# B&R Automation Studio project CoffeeMachine
Automation Studio 4.12.3.127 SP; Default project; technology packages: Acp10Arnc0 5.16.2, mappSafety 5.16.0, mappView 5.16.1

## Configuration ARX

CPU 4PPC30.043F-22B, AutomationRuntime B4.93, Build 4.1.2, Vc V4.72.6

### Hardware
```
4PPC30_043F_22B : 4PPC30.043F-22B v1.1.3.0
  Connector IF3:
    ActivateDevice = 1
  ConfigurationID = CoffeeMachine_ARX
  TimerDeviceType = SWIOTIMER
  Cyclic1Duration = 10000
  Cyclic1Tolerance = 10000
  Cyclic2Duration = 20000
  Cyclic2Tolerance = 20000
  Cyclic3Duration = 50000
  Cyclic3Tolerance = 50000
  Cyclic4Duration = 100000
  Cyclic4Tolerance = 100000
  Cyclic5Duration = 200000
  Cyclic5Tolerance = 200000
  Cyclic6Duration = 500000
  Cyclic6Tolerance = 500000
  Cyclic7Duration = 1000000
  Cyclic7Tolerance = 1000000
  Cyclic8Duration = 10000
  Cyclic8Tolerance = 30000000
  FileDevice1
  FileDeviceName1 = USER
  FileDevicePath1 = USER_PATH
  KeyMappingFile = VC\4PPC30_043F_22B.dis
```

## Configuration Simulation

CPU , AutomationRuntime B4.93, Build 4.1.2, Safety 0.0, Vc V4.72.6

### Hardware
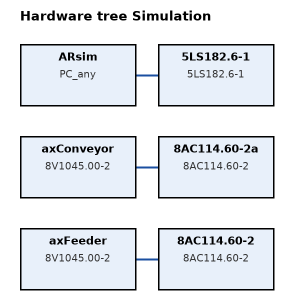
```
5LS182.6-1 : 5LS182.6-1 v1.3.1.0  [SL -> ARsim.SL1]
  Connector IF1:
    DNAConfiguration = manual
8AC114.60-2 : 8AC114.60-2 v1.0.0.8  [SS -> axFeeder.SS1; PLK1 -> 5LS182.6-1.IF1 (NodeNumber=1) [Cable Type=PowerlinkCable, Length=10, Version=1.0.0.3]; PLK2 -> 8AC114.60-2a.PLK1 (NodeNumber=1) [Cable Type=PowerlinkCable, Length=10, Version=1.0.0.3]]
8AC114.60-2a : 8AC114.60-2 v1.0.0.8  [SS -> axConveyor.SS1; PLK1 -> 8AC114.60-2.PLK2 (NodeNumber=2) [Cable Type=PowerlinkCable, Length=10, Version=1.0.0.3]]
ARsim : PC_any v1.1.1.0 (OrderNumber=PC)
  Connector IF3:
    Vnc1
    VncVcObjectName1 = Visu
    VncAuthentication1 = 1
    VncPasswordViewOnly1 = v
    VncPasswordViewControl1 = c
    VncRefreshRate1 = 200
    VncTitle1 = VNC - B&R Coffee Machine
  PreserveNonVolatileSystemSettings = 0
  BRObjects = 450
  XLinkUseDefault = 0
  Cyclic1Duration = 10000
  Cyclic1Tolerance = 0
  Cyclic2Duration = 200000
  Cyclic2Tolerance = 10000000
  Cyclic3Duration = 500000
  Cyclic3Tolerance = 10000000
  Cyclic4Duration = 1000000
  Cyclic4Tolerance = 10000000
  Cyclic5Duration = 2000000
  Cyclic5Tolerance = 10000000
  Cyclic6Duration = 3000000
  Cyclic6Tolerance = 12000000
  Cyclic7Duration = 4000000
  Cyclic7Tolerance = 12000000
  Cyclic8Duration = 5000000
  Cyclic8Tolerance = 30000000
  EthernetHostName = AR000CoffeeMachine
  ActivateOpcUa = 1
axConveyor : 8V1045.00-2 v2.2.0.0
  Simulate = standard
axFeeder : 8V1045.00-2 v2.2.0.0
  Simulate = standard
```

## Configuration T50_X20CP1586mcSim

### Task classes (Cpu.sw)
```
Cyclic#1 (cycle 2000 us, tolerance 0 us):
  mainlogic <- mainlogic.prg
  feeder <- FeederArm.feeder.prg
  conveyor <- ConveyorBelt.conveyor.prg
  brewing <- BrewingAssembly.brewing.prg
  heating <- FlowHeater.heating.prg
Cyclic#4:
  visCtrl <- Visualisation.visCtrl.prg
  visAlarm <- Visualisation.visAlarm.prg
  visTrend <- Visualisation.visTrend.prg
DataObjects: regular <- Recipes.regular.dob, cappu <- Recipes.cappu.dob, espres <- Recipes.espres.dob, Acp10sys
NcDataObjects: acp_err <- FeederArm.acp_err.dob, motor_sim <- FeederArm.motor_sim.dob, motor_offi <- FeederArm.motor_office.dob, feed_ini <- FeederArm.feed_ini.dob, conv_ini <- ConveyorBelt.conv_ini.dob
VcDataObjects: VisuW <- Visualisation.VisuW.dob
Binaries: vccdt, vccbmp, vccgauge, vccline, vcfile, arial, arialxsr, vccstr, vcbclass, VisuW03, vccbtn, vcmgr, vcgclass, vcdsint, vcnet, vcchtml, vcclbox, vcshared, vccslider, arialbd, vcxml, vccnum, vcpdvnc, FWRules, VisuW02, vccalarm, visvc, vccurl, vccshape, vccbar, vcctext, vcpdsw, vcfntttf, vccovl, vcalarm, VisuW01, vcctrend, udbdef, vcdsloc, vcchspot, vcpfx20, vctcal, vcrt, TCData, vcpfar00, Acp10map, acp10cfg, arconfig, asfw, iomap, Role, ashwd, ashwac, sysconf, User
Libraries: Convert, Runtime, sys_lib, brsystem, Standard, AsString, DataObj, FileIO, operator, AsTime, CoffeeLib, Visapi, AsArSdm, AsArProf, powerlnk, vcresman, ashw, SfDomain, MpBase
```

### Hardware
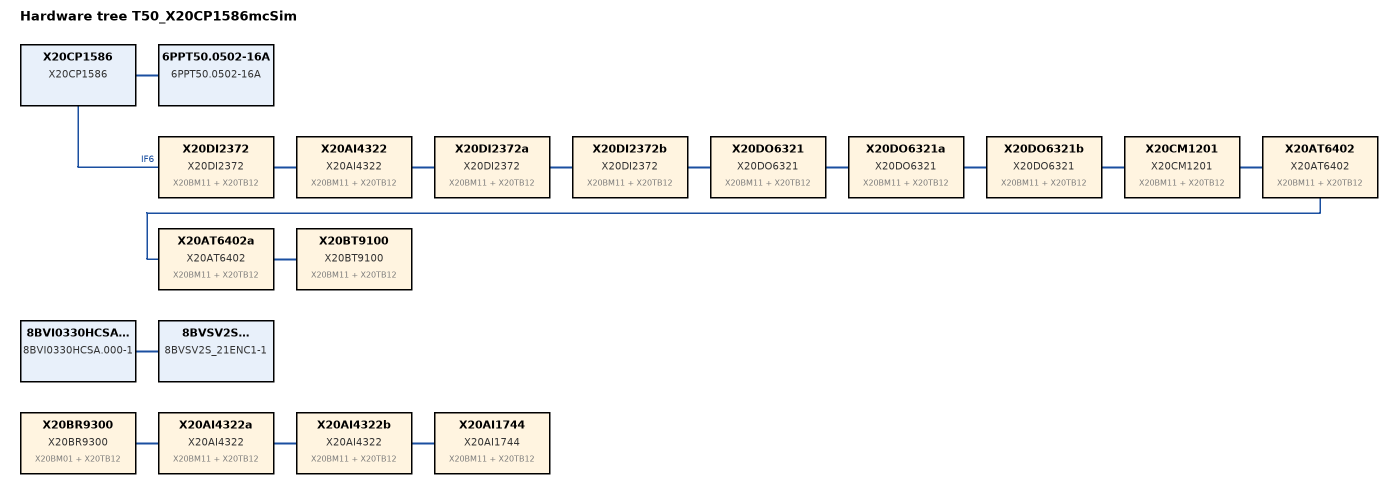
```
6PPT50.0502-16A : 6PPT50.0502-16A v1.3.8.0  [ETH2 -> X20CP1586.IF2 [Cable Type=PowerlinkCable, Length=10, Version=1.0.0.3]]
  Terminal = true
  PasswordVNC = 
  PasswordCIFS = 
  PasswordService = 
  VncVcObjectName = VisuW
  VncAuthentication = 1
  VncPasswordViewOnly = v
  VncPasswordViewControl = c
8BVI0330HCSA.000-1 : 8BVI0330HCSA.000-1 v2.3.0.1
  MotionTP = Acp10Arnc0
8BVSV2S_21ENC1-1 : 8BVSV2S_21ENC1-1 v2.4.0.0  [SS -> 8BVI0330HCSA.000-1.SS1]
X20AI1744 : X20AI1744 v1.10.0.0  [SS1 -> X20TB12o.SS; SL -> X20BM11m.SL1]
  Supervision = off
X20AI4322 : X20AI4322 v1.2.0.0  [SS1 -> X20TB12b.SS; SL -> X20BM11a.SL1]
  Supervision = off
X20AI4322a : X20AI4322 v1.2.0.0  [SS1 -> X20TB12m.SS; SL -> X20BM11k.SL1]
  Supervision = off
X20AI4322b : X20AI4322 v1.2.0.0  [SS1 -> X20TB12n.SS; SL -> X20BM11l.SL1]
  Supervision = off
X20AT6402 : X20AT6402 v1.2.0.0  [SS1 -> X20TB12i.SS; SL -> X20BM11h.SL1]
  Supervision = off
X20AT6402a : X20AT6402 v1.2.0.0  [SS1 -> X20TB12j.SS; SL -> X20BM11i.SL1]
  Supervision = off
X20BM01 : X20BM01 v2.2.0.0
X20BM11 : X20BM11 v1.1.0.0  [X2X1 -> X20CP1586.IF6]
X20BM11a : X20BM11 v1.1.0.0  [X2X1 -> X20BM11.X2X2]
X20BM11b : X20BM11 v1.1.0.0  [X2X1 -> X20BM11a.X2X2]
X20BM11c : X20BM11 v1.1.0.0  [X2X1 -> X20BM11b.X2X2]
X20BM11d : X20BM11 v1.1.0.0  [X2X1 -> X20BM11c.X2X2]
X20BM11e : X20BM11 v1.1.0.0  [X2X1 -> X20BM11d.X2X2]
X20BM11f : X20BM11 v1.1.0.0  [X2X1 -> X20BM11e.X2X2]
X20BM11g : X20BM11 v1.1.0.0  [X2X1 -> X20BM11f.X2X2]
X20BM11h : X20BM11 v1.1.0.0  [X2X1 -> X20BM11g.X2X2]
X20BM11i : X20BM11 v1.1.0.0  [X2X1 -> X20BM11h.X2X2]
X20BM11j : X20BM11 v1.1.0.0  [X2X1 -> X20BM11i.X2X2]
X20BM11k : X20BM11 v1.1.0.0  [X2X1 -> X20BM01.X2X2]
X20BM11l : X20BM11 v1.1.0.0  [X2X1 -> X20BM11k.X2X2]
X20BM11m : X20BM11 v1.1.0.0  [X2X1 -> X20BM11l.X2X2]
X20BR9300 : X20BR9300 v1.3.0.0  [SS1 -> X20TB12l.SS; SL -> X20BM01.SL1; X2X1 -> X20BT9100.X2X1 [Cable Type=X2XCable, Length=10, Version=1.0.0.3]]
  Supervision = off
X20BT9100 : X20BT9100 v1.3.0.0  [SS1 -> X20TB12k.SS; SL -> X20BM11j.SL1]
  Supervision = off
X20CM1201 : X20CM1201 v1.2.0.0  [SS1 -> X20TB12h.SS; SL -> X20BM11g.SL1]
  Supervision = off
X20CP1586 : X20CP1586 v1.10.0.0
  Connector IF2:
    ActivateDevice = 1
    HostName = br-automation_coffeemachine
  Connector IF3:
    DNAConfiguration = manual
    EplHostName = br-automation_coffeemachine
    HostName = br-automation_coffeemachine
  ConfigurationID = CoffeeMachine_T50_X20CP1586
  Simulation = 1
  Cyclic1Duration = 2000
  Cyclic1Tolerance = 0
  FileDevice1
  FileDeviceName1 = USER
  FileDevicePath1 = USER_PATH
  EthernetHostName = br-automation_coffeemachine
  ActivateDns = 1
X20DI2372 : X20DI2372 v1.2.0.0  [SS1 -> X20TB12a.SS; SL -> X20BM11.SL1]
  Supervision = off
X20DI2372a : X20DI2372 v1.2.0.0  [SS1 -> X20TB12c.SS; SL -> X20BM11b.SL1]
  Supervision = off
X20DI2372b : X20DI2372 v1.2.0.0  [SS1 -> X20TB12d.SS; SL -> X20BM11c.SL1]
  Supervision = off
X20DO6321 : X20DO6321 v1.2.0.0  [SS1 -> X20TB12e.SS; SL -> X20BM11d.SL1]
  Supervision = off
X20DO6321a : X20DO6321 v1.2.0.0  [SS1 -> X20TB12f.SS; SL -> X20BM11e.SL1]
  Supervision = off
X20DO6321b : X20DO6321 v1.2.0.0  [SS1 -> X20TB12g.SS; SL -> X20BM11f.SL1]
  Supervision = off
X20TB12a : X20TB12 v1.0.0.0
X20TB12b : X20TB12 v1.0.0.0
X20TB12c : X20TB12 v1.0.0.0
X20TB12d : X20TB12 v1.0.0.0
X20TB12e : X20TB12 v1.0.0.0
X20TB12f : X20TB12 v1.0.0.0
X20TB12g : X20TB12 v1.0.0.0
X20TB12h : X20TB12 v1.0.0.0
X20TB12i : X20TB12 v1.0.0.0
X20TB12j : X20TB12 v1.0.0.0
X20TB12k : X20TB12 v1.0.0.0
X20TB12l : X20TB12 v1.0.0.0
X20TB12m : X20TB12 v1.0.0.0
X20TB12n : X20TB12 v1.0.0.0
X20TB12o : X20TB12 v1.0.0.0
```

### IoMap.iom - X20CP1586/IoMap.iom
```iecst
VAR_CONFIG
	Cyclic#1.::doDoseCoffee AT %QX."X20DO6321".DigitalOutput05;
END_VAR
```

## Logical view

Binary libraries used (declarations not repeated): Convert, Runtime, sys_lib, brsystem, Standard, AsString, DataObj, FileIO, operator, AsTime, CoffeeLib, Visapi, AsArSdm, AsArProf, LoopConR, Acp10man, Acp10par, NcGlobal, Acp10sim, Acp10_MC, Acp10sdc, SfDomain, MpBase

### Global.var - Global Variables
```iecst
(********************************************************************
 * COPYRIGHT -- B&R
 ********************************************************************
 * File: Global.var
 * Author: B&R
 * Created: June 06, 2007
 ********************************************************************
 * Global variables of project coffee
 ********************************************************************)
VAR
	axFeeder : ACP10AXIS_typ; (*axis information of feeder*)
	axConveyor : ACP10AXIS_typ; (*axis information of conveyor*)
	doCupPull : BOOL := FALSE; (*pulls cup out of storage*)
	gMainLogic : main_typ; (*info structure of main logic*)
	gFeeder : feeder_typ := (0); (*info structure of feeder*)
	gBrewing : brewing_typ := (0); (*info structure of brewing assembly*)
	doDoseMilk : BOOL := FALSE; (*doser: milk*)
	doDoseSugar : BOOL := FALSE; (*doser: sugar*)
	doDoseCoffee : BOOL := FALSE; (*doser: coffee*)
	gConveyor : conveyor_typ := (0);
	gHeating : heating_typ := (0); (*info structure of heating*)
	doPumpWater : BOOL := FALSE; (*water pump*)
	aoHeating : INT := 0; (*heating control*)
	atWaterTemp : INT := 0; (*actual temperature of water*)
	diStart_Coffee : BOOL := FALSE; (*start making coffee*)
	gActConveyorVelocity : REAL; (*actual conveyor velocity*)
	gActFeederVelocity : REAL; (*actual feeder velocity*)
	gActFeederPosition : REAL; (*actual feeder position*)
	gActConveyorPosition : REAL; (*actual conveyor position*)
END_VAR
```

### Package Logical/BrewingAssembly - Brewing & Dosing

### Program Logical/BrewingAssembly/brewing

#### brewing.var
```iecst
(********************************************************************
 * COPYRIGHT -- B&R
 ********************************************************************
 * Package: Brewing
 * File: brewing.var
 * Author: B&R
 * Created: June 14, 2007
 *******************************************************************)
VAR
	pBrewingText_ : UDINT := 0;
END_VAR
VAR CONSTANT
	sSTANDBY : UINT := 0;
	sDOSING : UINT := 10;
	sBREWING : UINT := 20;
	sFINISH : UINT := 30;
END_VAR
VAR
	milkTP : TP;
	coffeeTP : TP;
	sugarTP : TP;
	waterTP : TP;
END_VAR
```

#### brewing.st
```iecst
(********************************************************************
 * COPYRIGHT -- B&R
 ********************************************************************
 * Program: Brewing
 * File: Brewing.st
 * Author: B&R
 * Created: June 12, 2007
 ********************************************************************
 * Implementation of program Brewing
 ********************************************************************)

PROGRAM _CYCLIC
	(* plain text information of current step *)
	IF (pBrewingText_ <> 0) THEN
			strcpy(ADR(gBrewing.status.brewingStepText), pBrewingText_);
	END_IF

	IF EDGEPOS(diStart_Coffee1) = TRUE THEN
 		gMainLogic.status.progressStep := 0;			(* transporting cup to brewing station *)
	END_IF

	CASE gBrewing.status.sBrewingStep OF
		(* wait for start signal *)
		sSTANDBY:
			pBrewingText_ := ADR('sSTANDBY');

			IF (gBrewing.cmd.start = TRUE) THEN
				gMainLogic.status.progressStep := 1;			(* brewing in progress *)
   			    gBrewing.cmd.start   := FALSE;
				gBrewing.status.done := FALSE;
				gBrewing.status.sBrewingStep := sDOSING;
			END_IF

		(* dose ingredients according to recipe *)
		sDOSING:
			pBrewingText_ := ADR('sDOSING');

			milkTP  (IN := 1, PT := REAL_TO_TIME(gMainLogic.par.recipe.milk   * 10));	(* 100ml -> 1s *)
			sugarTP (IN := 1, PT := REAL_TO_TIME(gMainLogic.par.recipe.sugar  * 10));  (* 50g -> 500ms *)
			coffeeTP(IN := 1, PT := REAL_TO_TIME(gMainLogic.par.recipe.coffee * 10));  (* 80g -> 800ms *)

			doDoseMilk   := milkTP.Q;
			doDoseSugar  := sugarTP.Q;
			doDoseCoffee := coffeeTP.Q;

			(* wait until dosing is finished *)
			IF (milkTP.Q = 0) AND (sugarTP.Q = 0) AND (coffeeTP.Q = 0) THEN
				milkTP  (IN := 0, PT := 0);
				sugarTP (IN := 0, PT := 0);
				coffeeTP(IN := 0, PT := 0);
	 			gBrewing.status.sBrewingStep := sBREWING;
	 		END_IF

		(* brew coffee *)
		sBREWING:
			pBrewingText_ := ADR('sBREWING');

			(* start brewing if set temperature has been reached *)
			IF (gHeating.status.setTempOK = TRUE) THEN
				waterTP(IN := 1, PT := REAL_TO_TIME(gMainLogic.par.recipe.water * 50));		(* 100ml -> 1s *)

				doPumpWater := waterTP.Q;

				(* wait until dosing is finished *)
				IF (waterTP.Q = 0) THEN
					waterTP(IN := 0, PT := 0);
		 			gBrewing.status.sBrewingStep := sFINISH;
		 		END_IF
			END_IF

		(* all done *)
		sFINISH:
			pBrewingText_ := ADR('sFINISH');

			gMainLogic.status.progressStep := 2;			(* ready for take out *)

			gBrewing.status.done := TRUE;
			gBrewing.status.sBrewingStep := sSTANDBY;
	END_CASE;
END_PROGRAM
```

- Visualisation Logical/Visualisation (not shown)

### Package Logical/Libraries - Global Libraries

- Visualisation Logical/mappView (not shown)

Listed in the project but not available here: Logical/Doc, Logical/Global.typ, Logical/mainlogic, Logical/ConveyorBelt, Logical/FeederArm, Logical/FlowHeater, Logical/Recipes
